// TIA Portal V19 export
DATA_BLOCK "SET PARAMETER DB"   // DB7
{ S7_Optimized_Access := 'TRUE' }
// stored: MemoryReserve 100
   VAR
      "MANUAL VFD SET PARAMETER" : Struct
         "MFG VESSEL MOTOR SPEED" : Real;
         "PREMIXING VESSEL MOTOR SPEED" : Real;
         "STORAGE VESSEL-1 MOTOR SPEED" : Real;
         "STORAGE VESSEL-2 MOTOR SPEED" : Real;
         "SUGAR VESSEL MOTOR SPEED" : Real;
         "AO SPARE_1" : Real;
         "AO SPARE_2" : Real;
         "AO SPARE_3" : Real;
      END_STRUCT;
      "AUTO VFD SET PARAMETER" : Struct
         "MFG VESSEL MOTOR SPEED" : Real;
         "PREMIXING VESSEL MOTOR SPEED" : Real;
         "STORAGE VESSEL-1 MOTOR SPEED" : Real;
         "STORAGE VESSEL-2 MOTOR SPEED" : Real;
         "SUGAR VESSEL MOTOR SPEED" : Real;
         "AO SPARE_1" : Real;
         "AO SPARE_2" : Real;
         "AO SPARE_3" : Real;
      END_STRUCT;
   END_VAR
BEGIN
END_DATA_BLOCK
